Staubli VAL3: tool.dtx

num nIndex
num nIndexTool
num nKey
public num nPage
num nRefresh
num nTime = 1
num nView
string sEvent
public string sItems
string sList
string sMenu
string sMessage
string sMenu8[8]
string sActionON[3]
string sActionOFF[3]
bool bButton[8]
bool bLarge
